Staubli VAL3: MsgTypeStaubli.pjx

--- MsgTypeStaubli.pjx ---
Parameters version=s7.8.1 stackSize=5000 millimeterUnit=true
Program file=start.pgx
Program file=stop.pgx
Data file=MsgTypeStaubli.dtx

--- MsgTypeStaubli.dtx ---
public num READ_IO
public num SET_DRIVE_POWER
public num VELOCITY_CFG
public num VELOCITY_CMD
public num WRITE_SINGLE_IO
